FUNCTION_BLOCK  TcoEcatSlaveState EXTENDS TcoObject 
VAR_INPUT
    AdsAddr : AMSADDR;
END_VAR
VAR_OUTPUT
END_VAR
VAR

    //*	{attribute addProperty Name "<#Actual state#>"}
    //*	{attribute clr [ReadOnly()]}
    _ecatState : eEcatState;
    //*	{attribute addProperty Name "<#Actual Link state#>"}
    //*	{attribute clr [ReadOnly()]}
    _linkState : eLinkState;
    //*	{attribute addProperty Name "<#ECAT Communication Ok#>"}
    //*	{attribute clr [ReadOnly()]}
    _ecatOk : BOOL;
 
    //*	{attribute clr [RenderIgnore()]}
    _progress : INT := 0;
	

    //*	{attribute addProperty Name "<#EtherCat masters Ams Net Id#>"}
    //*	{attribute clr [ReadOnly()]}
    _netId : STRING[23]; //as string	

	 //* {attribute clr [RenderIgnore()]}
    _etherCAT_Addr : UINT;

	//*	{attribute addProperty Name "<#State check Time(Period)#>"}
   	_periodStateCheckTime: TIME :=T#1S;
	
	//*	{attribute addProperty Name "<#Error Time#>"}
   	_errorTime: TIME :=T#5S;
    //*	{attribute clr [RenderIgnore()]}
    _getSlaveState : FB_EcGetSlaveState;
    //*	{attribute clr [RenderIgnore()]}
    _setSlaveState : FB_EcSetSlaveState;


    //*	{attribute clr [RenderIgnore()]}
    bExecute : BOOL;
    //*	{attribute clr [RenderIgnore()]}
    state : ST_EcSlaveState;
    //*	{attribute clr [RenderIgnore()]}
    _error : BOOL;
    //*	{attribute clr [RenderIgnore()]}
    _busy : BOOL;
    //*	{attribute clr [RenderIgnore()]}
    _errId : UDINT;
    //*	{attribute clr [RenderIgnore()]}
    _stateTimer : TON;
	//*	{attribute clr [RenderIgnore()]}
    _errorTimer : TON;
	
    //*	{attribute addProperty Name "<#Required state#>"}
    _ecatReqestState : eEcatState;
	
    //*	{attribute addProperty Name "<#Change State#>"}
    _changeStateTask : TcoCore.TcoTask(THIS^);

    //*	{attribute addProperty Name "<#Restore#>"}
    _restoreTask : TcoCore.TcoTask(THIS^);

	 {attribute 'hide'} 
	_sb : TcoCore.StringBuilder;
	{attribute 'hide'} 
	_amsEmpty: BOOL;
END_VAR

_netId := F_CreateAmsNetId(nIds := AdsAddr.netId);
_etherCAT_Addr := AdsAddr.port;
_amsEmpty:=(_netId = '0.0.0.0.0.0') OR (_etherCAT_Addr = 0);
	

IF _changeStateTask.Execute() THEN
	_changeStateTask.DoneWhen(ChangeState(RequestedDeviceState:=_ecatReqestState ));
END_IF

THIS^._changeStateTask.ThrowWhen((_changeStateTask.ElapsedTime>=_errorTime AND _progress>0) 
								OR _amsEmpty ); 

THIS^._changeStateTask.Messenger.OnCondition(_amsEmpty).Error('<#Ads address information is not defined!#>');
//*************RESTORE********************

_restoreTask.Enabled := TRUE;
IF _restoreTask.Execute() THEN
	Restore();
END_IF
//****************************************


IF (_amsEmpty) THEN		
	RETURN;
END_IF


THIS^._GetState(_periodStateCheckTime);

METHOD PRIVATE _GetState
VAR_INPUT
	Period:TIME;
END_VAR
_stateTimer(IN := TRUE,PT := Period);		

IF _stateTimer.Q THEN
	bExecute := TRUE;
	_stateTimer(IN := FALSE);
END_IF
 
_getSlaveState(sNetId:= _netId, 
				nSlaveAddr := _etherCAT_Addr, 
				bExecute := bExecute,
				bBusy => _busy,
				state => state,
				bError => _error,
				nErrId => _ErrId);

IF NOT _busy THEN
	_ecatState := state.deviceState;
	_linkState := state.linkState;
	_ecatOk := (state.deviceState = EC_DEVICE_STATE_OP);
	bExecute := FALSE;
END_IF
END_METHOD

PROPERTY PUBLIC EcatOk : BOOL
GET
EcatOk:=_ecatOk;
END_GET
END_PROPERTY

PROPERTY PUBLIC ErrorTime : TIME
GET
ErrorTime:=_errorTime;
END_GET
SET
_errorTime:=ErrorTime;
END_SET
END_PROPERTY

METHOD PUBLIC ChangeState : BOOL
VAR_INPUT
	RequestedDeviceState:BYTE;
END_VAR
ChangeState := FALSE;

_setSlaveState(sNetId := _netId,
    nSlaveAddr := _etherCAT_Addr,
    bExecute :=,
    tTimeout :=,
    reqState :=,
    bBusy =>,
    bError =>,
    nErrId =>,
    currState => state);

CASE _progress OF
    0:
        _ecatOk := FALSE;
        _setSlaveState(bExecute := FALSE);
        _progress := 10;

    10:
        _setSlaveState(reqState := EC_DEVICE_STATE_INIT);
        _setSlaveState(bExecute := TRUE);

        IF _setSlaveState.bBusy THEN
            _progress := 15;
        END_IF
    15: //INIT
        IF (state.deviceState) = EC_DEVICE_STATE_INIT AND
            RequestedDeviceState > state.deviceState AND
            RequestedDeviceState <> EC_DEVICE_STATE_BOOTSTRAP THEN
            _setSlaveState(bExecute := FALSE);
            _progress := 30;
        ELSIF (state.deviceState) = EC_DEVICE_STATE_INIT AND
            RequestedDeviceState > state.deviceState AND
            RequestedDeviceState = EC_DEVICE_STATE_BOOTSTRAP THEN
            _setSlaveState(bExecute := FALSE);
            _progress := 20;
        ELSIF NOT _setSlaveState.bBusy AND (state.deviceState) = RequestedDeviceState THEN
            _progress := 100;

        END_IF

    20:
        _setSlaveState(reqState := EC_DEVICE_STATE_BOOTSTRAP);
        _setSlaveState(bExecute := TRUE);

        IF _setSlaveState.bBusy THEN
            _progress := 25;
        END_IF
    25: ///BOOTSTRAP
        IF (state.deviceState) = EC_DEVICE_STATE_BOOTSTRAP THEN
            _setSlaveState(bExecute := FALSE);
            _progress := 100;
        END_IF

    30:
        _setSlaveState(reqState := EC_DEVICE_STATE_PREOP);
        _setSlaveState(bExecute := TRUE);

        IF _setSlaveState.bBusy THEN
            _progress := 35;
        END_IF
    35: //PREOP
        IF (state.deviceState) = EC_DEVICE_STATE_PREOP AND RequestedDeviceState > state.deviceState THEN
            _setSlaveState(bExecute := FALSE);
            _progress := 40;
        ELSIF NOT _setSlaveState.bBusy AND (state.deviceState) = RequestedDeviceState THEN
            _progress := 100;
        END_IF

    40:
        _setSlaveState(reqState := EC_DEVICE_STATE_SAFEOP);
        _setSlaveState(bExecute := TRUE);

        IF _setSlaveState.bBusy THEN
            _progress := 45;
        END_IF
    45: //SAFEOP
        IF (state.deviceState) = EC_DEVICE_STATE_SAFEOP AND RequestedDeviceState > state.deviceState THEN
            _setSlaveState(bExecute := FALSE);
            _progress := 50;
        ELSIF NOT _setSlaveState.bBusy AND (state.deviceState) = RequestedDeviceState THEN
            _progress := 100;
        END_IF

    50: //OP
        _setSlaveState(reqState := EC_DEVICE_STATE_OP);
        _setSlaveState(bExecute := TRUE);

        IF (state.deviceState) = EC_DEVICE_STATE_OP THEN
            _setSlaveState(bExecute := FALSE);
            _ecatOk := TRUE;
            _progress := 100;

        END_IF

    100:

        ChangeState := TRUE;
        _progress := 0;

END_CASE
Messenger.OnCondition(NOT _setSlaveState.bBusy AND RequestedDeviceState > EC_DEVICE_STATE_OP)
    .Post(_sb.Clear().Append('<#Unexpected state: #>').Append(TO_STRING(state.deviceState)).ToString(), eMessageCategory.Error);
END_METHOD

PROPERTY PUBLIC ChangeStateTask : TcoCore.ITcoTaskStatus
GET
ChangeStateTask:=_changeStateTask;
END_GET
END_PROPERTY

PROPERTY PUBLIC PeriodCheckState : TIME
GET
PeriodCheckState:= _periodStateCheckTime;
END_GET
SET
_periodStateCheckTime:=PeriodCheckState;
END_SET
END_PROPERTY

METHOD Restore  : ITcoRestorable
VAR_INPUT
END_VAR
_changeStateTask.Restore();
_ecatOk:=false;
_progress:=0;
_restoreTask.Restore();
END_METHOD

END_FUNCTION_BLOCK

(* stored: Version 1.1.0.1, ProductVersion 3.1.4024.11
   POU TcoEcatSlaveState: Id {5035a144-a13f-0775-217b-e1425fee930c}, SpecialFunc None
   Folder Internal: Id {a2e5e2ee-1878-07e8-1f6d-0423d58d8da9}
   Folder Public: Id {093f1a08-c90b-0553-3579-1779a2c8bb6b}
   Method _GetState: Id {5814f303-9529-0909-235f-53a111b03cf0}
   Property EcatOk: Id {c55e70fb-51cf-0b56-1481-6f363db4f440}
   Get Get: Id {047e20bc-f624-0618-3d51-5a57753e58de}
   Property ErrorTime: Id {c3f135ca-ccd1-0200-3f6c-495a9ee20275}
   Get Get: Id {e82ab372-955d-0a1b-3c81-28905b737981}
   Set Set: Id {d8909174-7c04-0e77-13f5-17ccdf218cc4}
   Method ChangeState: Id {3b8371cc-b5cf-0927-320c-caa7528b1d35}
   Property ChangeStateTask: Id {ccae978c-c808-0249-24be-69f5c64b4959}
   Get Get: Id {3b18ffe4-915b-0d73-15e6-481ccf859b65}
   Property PeriodCheckState: Id {9eb45a84-7e27-03dd-1f9e-9ef82f5302f1}
   Get Get: Id {95709821-c07d-067e-2643-2f586889bbc3}
   Set Set: Id {239a42eb-b878-05ee-1163-39f86025e757}
   Method Restore: Id {0fe634ae-4b55-037f-150d-2d2eb2241799} *)
